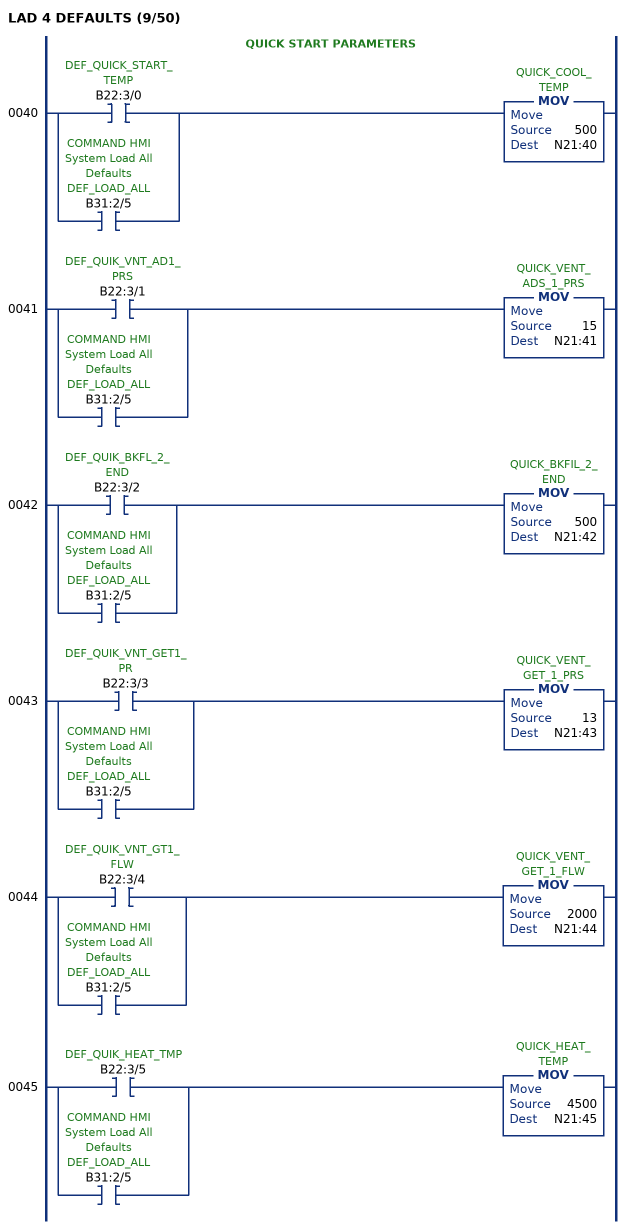
% Rung: 40 %
% TITLE: QUICK START PARAMETERS %
SOR BST XIC B22:3/0 NXB XIC B31:2/5 BND MOV 500 N21:40 EOR
%   B22:3/0  DEF_QUICK_START_TEMP %
%   B31:2/5  DEF_LOAD_ALL  "COMMAND HMI System Load All Defaults" %
%   N21:40  QUICK_COOL_TEMP %
% Rung: 41 %
SOR BST XIC B22:3/1 NXB XIC B31:2/5 BND MOV 15 N21:41 EOR
%   B22:3/1  DEF_QUIK_VNT_AD1_PRS %
%   B31:2/5  DEF_LOAD_ALL  "COMMAND HMI System Load All Defaults" %
%   N21:41  QUICK_VENT_ADS_1_PRS %
% Rung: 42 %
SOR BST XIC B22:3/2 NXB XIC B31:2/5 BND MOV 500 N21:42 EOR
%   B22:3/2  DEF_QUIK_BKFL_2_END %
%   B31:2/5  DEF_LOAD_ALL  "COMMAND HMI System Load All Defaults" %
%   N21:42  QUICK_BKFIL_2_END %
% Rung: 43 %
SOR BST XIC B22:3/3 NXB XIC B31:2/5 BND MOV 13 N21:43 EOR
%   B22:3/3  DEF_QUIK_VNT_GET1_PR %
%   B31:2/5  DEF_LOAD_ALL  "COMMAND HMI System Load All Defaults" %
%   N21:43  QUICK_VENT_GET_1_PRS %
% Rung: 44 %
SOR BST XIC B22:3/4 NXB XIC B31:2/5 BND MOV 2000 N21:44 EOR
%   B22:3/4  DEF_QUIK_VNT_GT1_FLW %
%   B31:2/5  DEF_LOAD_ALL  "COMMAND HMI System Load All Defaults" %
%   N21:44  QUICK_VENT_GET_1_FLW %
% Rung: 45 %
SOR BST XIC B22:3/5 NXB XIC B31:2/5 BND MOV 4500 N21:45 EOR
%   B22:3/5  DEF_QUIK_HEAT_TMP %
%   B31:2/5  DEF_LOAD_ALL  "COMMAND HMI System Load All Defaults" %
%   N21:45  QUICK_HEAT_TEMP %

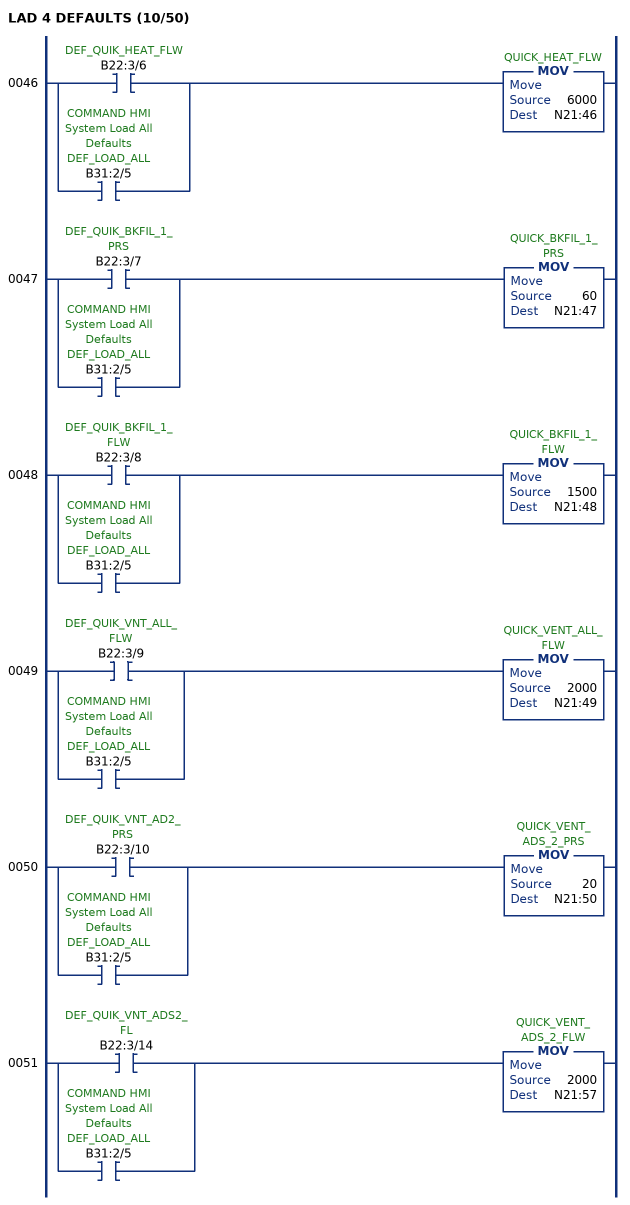
% Rung: 46 %
SOR BST XIC B22:3/6 NXB XIC B31:2/5 BND MOV 6000 N21:46 EOR
%   B22:3/6  DEF_QUIK_HEAT_FLW %
%   B31:2/5  DEF_LOAD_ALL  "COMMAND HMI System Load All Defaults" %
%   N21:46  QUICK_HEAT_FLW %
% Rung: 47 %
SOR BST XIC B22:3/7 NXB XIC B31:2/5 BND MOV 60 N21:47 EOR
%   B22:3/7  DEF_QUIK_BKFIL_1_PRS %
%   B31:2/5  DEF_LOAD_ALL  "COMMAND HMI System Load All Defaults" %
%   N21:47  QUICK_BKFIL_1_PRS %
% Rung: 48 %
SOR BST XIC B22:3/8 NXB XIC B31:2/5 BND MOV 1500 N21:48 EOR
%   B22:3/8  DEF_QUIK_BKFIL_1_FLW %
%   B31:2/5  DEF_LOAD_ALL  "COMMAND HMI System Load All Defaults" %
%   N21:48  QUICK_BKFIL_1_FLW %
% Rung: 49 %
SOR BST XIC B22:3/9 NXB XIC B31:2/5 BND MOV 2000 N21:49 EOR
%   B22:3/9  DEF_QUIK_VNT_ALL_FLW %
%   B31:2/5  DEF_LOAD_ALL  "COMMAND HMI System Load All Defaults" %
%   N21:49  QUICK_VENT_ALL_FLW %
% Rung: 50 %
SOR BST XIC B22:3/10 NXB XIC B31:2/5 BND MOV 20 N21:50 EOR
%   B22:3/10  DEF_QUIK_VNT_AD2_PRS %
%   B31:2/5  DEF_LOAD_ALL  "COMMAND HMI System Load All Defaults" %
%   N21:50  QUICK_VENT_ADS_2_PRS %
% Rung: 51 %
SOR BST XIC B22:3/14 NXB XIC B31:2/5 BND MOV 2000 N21:57 EOR
%   B22:3/14  DEF_QUIK_VNT_ADS2_FL %
%   B31:2/5  DEF_LOAD_ALL  "COMMAND HMI System Load All Defaults" %
%   N21:57  QUICK_VENT_ADS_2_FLW %

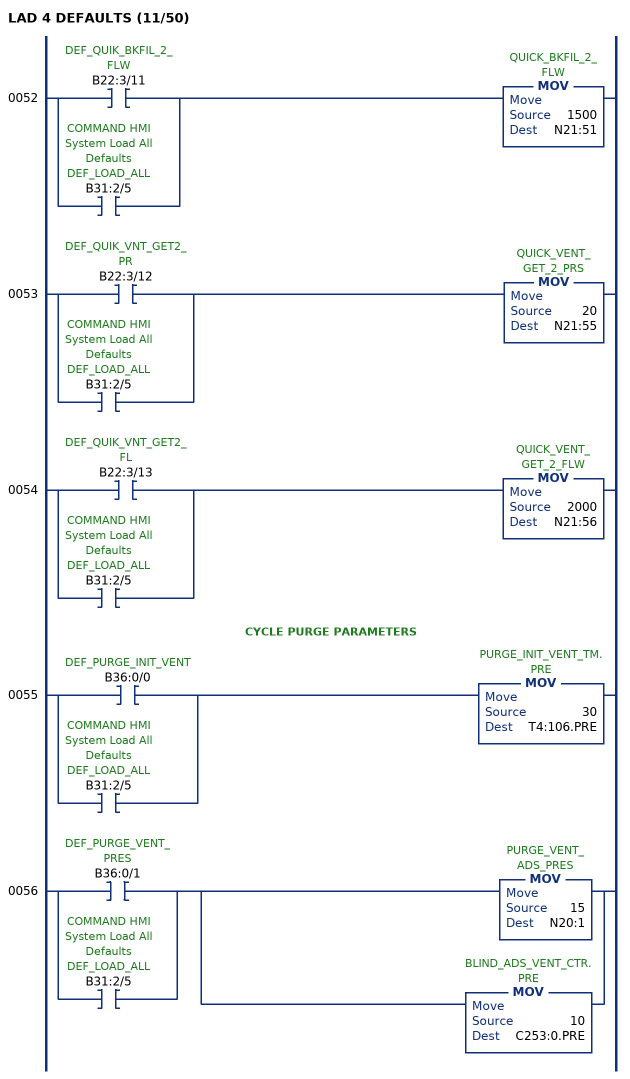
% Rung: 52 %
SOR BST XIC B22:3/11 NXB XIC B31:2/5 BND MOV 1500 N21:51 EOR
%   B22:3/11  DEF_QUIK_BKFIL_2_FLW %
%   B31:2/5  DEF_LOAD_ALL  "COMMAND HMI System Load All Defaults" %
%   N21:51  QUICK_BKFIL_2_FLW %
% Rung: 53 %
SOR BST XIC B22:3/12 NXB XIC B31:2/5 BND MOV 20 N21:55 EOR
%   B22:3/12  DEF_QUIK_VNT_GET2_PR %
%   B31:2/5  DEF_LOAD_ALL  "COMMAND HMI System Load All Defaults" %
%   N21:55  QUICK_VENT_GET_2_PRS %
% Rung: 54 %
SOR BST XIC B22:3/13 NXB XIC B31:2/5 BND MOV 2000 N21:56 EOR
%   B22:3/13  DEF_QUIK_VNT_GET2_FL %
%   B31:2/5  DEF_LOAD_ALL  "COMMAND HMI System Load All Defaults" %
%   N21:56  QUICK_VENT_GET_2_FLW %
% Rung: 55 %
% TITLE: CYCLE PURGE PARAMETERS %
SOR BST XIC B36:0/0 NXB XIC B31:2/5 BND MOV 30 T4:106.PRE EOR
%   B36:0/0  DEF_PURGE_INIT_VENT %
%   B31:2/5  DEF_LOAD_ALL  "COMMAND HMI System Load All Defaults" %
%   T4:106  PURGE_INIT_VENT_TM %
% Rung: 56 %
SOR BST XIC B36:0/1 NXB XIC B31:2/5 BND BST MOV 15 N20:1 NXB MOV 10 C253:0.PRE BND EOR
%   B36:0/1  DEF_PURGE_VENT_PRES %
%   B31:2/5  DEF_LOAD_ALL  "COMMAND HMI System Load All Defaults" %
%   N20:1  PURGE_VENT_ADS_PRES %
%   C253:0  BLIND_ADS_VENT_CTR %

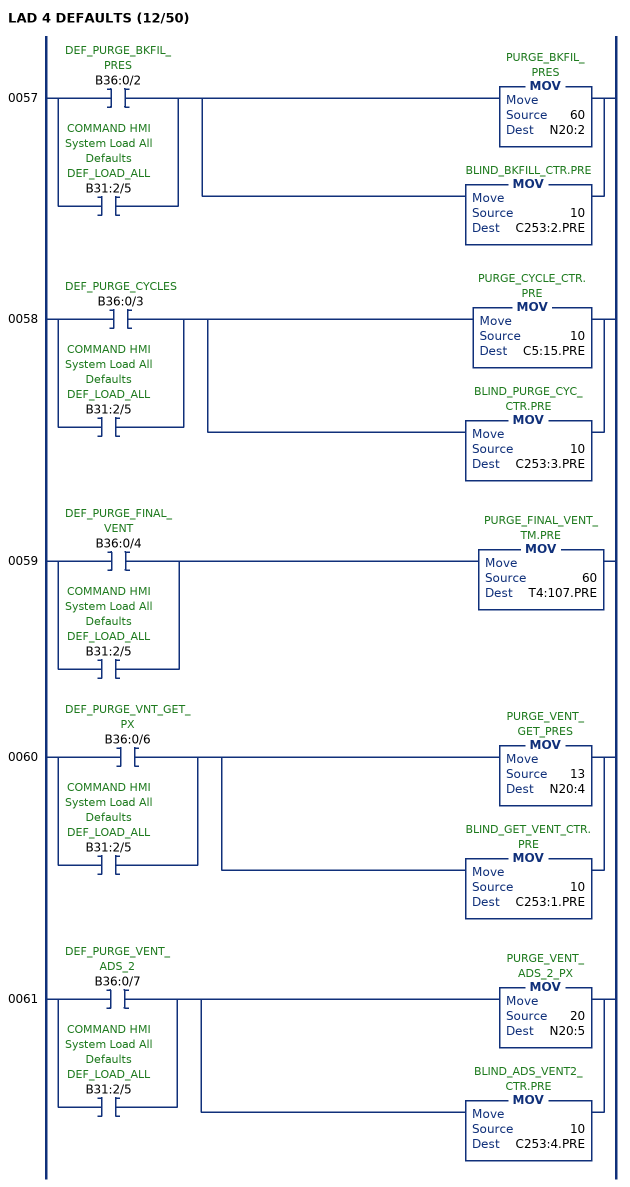
% Rung: 57 %
SOR BST XIC B36:0/2 NXB XIC B31:2/5 BND BST MOV 60 N20:2 NXB MOV 10 C253:2.PRE BND EOR
%   B36:0/2  DEF_PURGE_BKFIL_PRES %
%   B31:2/5  DEF_LOAD_ALL  "COMMAND HMI System Load All Defaults" %
%   N20:2  PURGE_BKFIL_PRES %
%   C253:2  BLIND_BKFILL_CTR %
% Rung: 58 %
SOR BST XIC B36:0/3 NXB XIC B31:2/5 BND BST MOV 10 C5:15.PRE NXB MOV 10 C253:3.PRE BND EOR
%   B36:0/3  DEF_PURGE_CYCLES %
%   B31:2/5  DEF_LOAD_ALL  "COMMAND HMI System Load All Defaults" %
%   C5:15  PURGE_CYCLE_CTR %
%   C253:3  BLIND_PURGE_CYC_CTR %
% Rung: 59 %
SOR BST XIC B36:0/4 NXB XIC B31:2/5 BND MOV 60 T4:107.PRE EOR
%   B36:0/4  DEF_PURGE_FINAL_VENT %
%   B31:2/5  DEF_LOAD_ALL  "COMMAND HMI System Load All Defaults" %
%   T4:107  PURGE_FINAL_VENT_TM %
% Rung: 60 %
SOR BST XIC B36:0/6 NXB XIC B31:2/5 BND BST MOV 13 N20:4 NXB MOV 10 C253:1.PRE BND EOR
%   B36:0/6  DEF_PURGE_VNT_GET_PX %
%   B31:2/5  DEF_LOAD_ALL  "COMMAND HMI System Load All Defaults" %
%   N20:4  PURGE_VENT_GET_PRES %
%   C253:1  BLIND_GET_VENT_CTR %
% Rung: 61 %
SOR BST XIC B36:0/7 NXB XIC B31:2/5 BND BST MOV 20 N20:5 NXB MOV 10 C253:4.PRE BND EOR
%   B36:0/7  DEF_PURGE_VENT_ADS_2 %
%   B31:2/5  DEF_LOAD_ALL  "COMMAND HMI System Load All Defaults" %
%   N20:5  PURGE_VENT_ADS_2_PX %
%   C253:4  BLIND_ADS_VENT2_CTR %

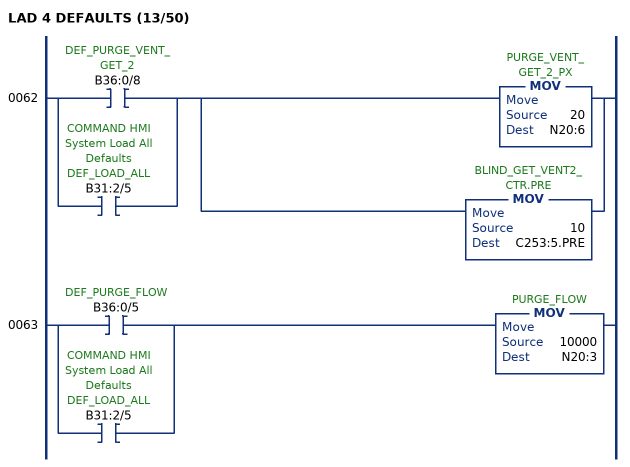
% Rung: 62 %
SOR BST XIC B36:0/8 NXB XIC B31:2/5 BND BST MOV 20 N20:6 NXB MOV 10 C253:5.PRE BND EOR
%   B36:0/8  DEF_PURGE_VENT_GET_2 %
%   B31:2/5  DEF_LOAD_ALL  "COMMAND HMI System Load All Defaults" %
%   N20:6  PURGE_VENT_GET_2_PX %
%   C253:5  BLIND_GET_VENT2_CTR %
% Rung: 63 %
SOR BST XIC B36:0/5 NXB XIC B31:2/5 BND MOV 10000 N20:3 EOR
%   B36:0/5  DEF_PURGE_FLOW %
%   B31:2/5  DEF_LOAD_ALL  "COMMAND HMI System Load All Defaults" %
%   N20:3  PURGE_FLOW %

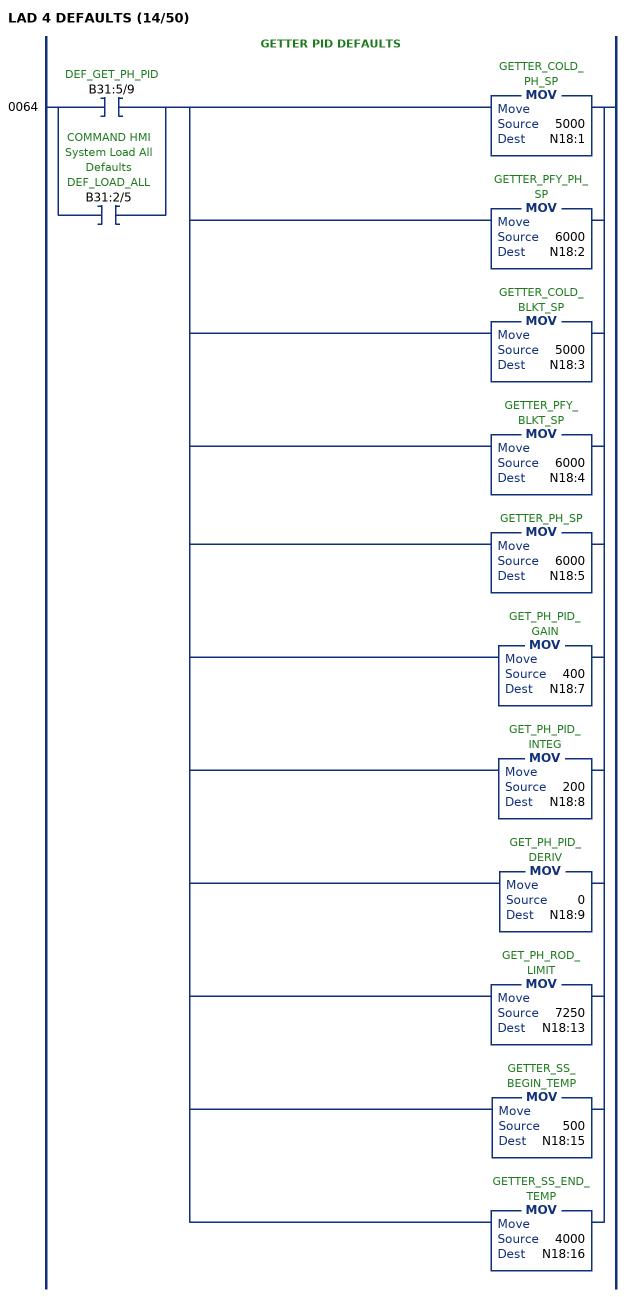
% Rung: 64 %
% TITLE: GETTER PID DEFAULTS %
SOR BST XIC B31:5/9 NXB XIC B31:2/5 BND BST MOV 5000 N18:1 NXB MOV 6000 N18:2 NXB MOV 5000 N18:3 NXB MOV 6000 N18:4 NXB MOV 6000 N18:5 NXB MOV 400 N18:7 NXB MOV 200 N18:8 NXB MOV 0 N18:9 NXB MOV 7250 N18:13 NXB MOV 500 N18:15 NXB MOV 4000 N18:16 BND EOR
%   B31:5/9  DEF_GET_PH_PID %
%   B31:2/5  DEF_LOAD_ALL  "COMMAND HMI System Load All Defaults" %
%   N18:1  GETTER_COLD_PH_SP %
%   N18:2  GETTER_PFY_PH_SP %
%   N18:3  GETTER_COLD_BLKT_SP %
%   N18:4  GETTER_PFY_BLKT_SP %
%   N18:5  GETTER_PH_SP %
%   N18:7  GET_PH_PID_GAIN %
%   N18:8  GET_PH_PID_INTEG %
%   N18:9  GET_PH_PID_DERIV %
%   N18:13  GET_PH_ROD_LIMIT %
%   N18:15  GETTER_SS_BEGIN_TEMP %
%   N18:16  GETTER_SS_END_TEMP %

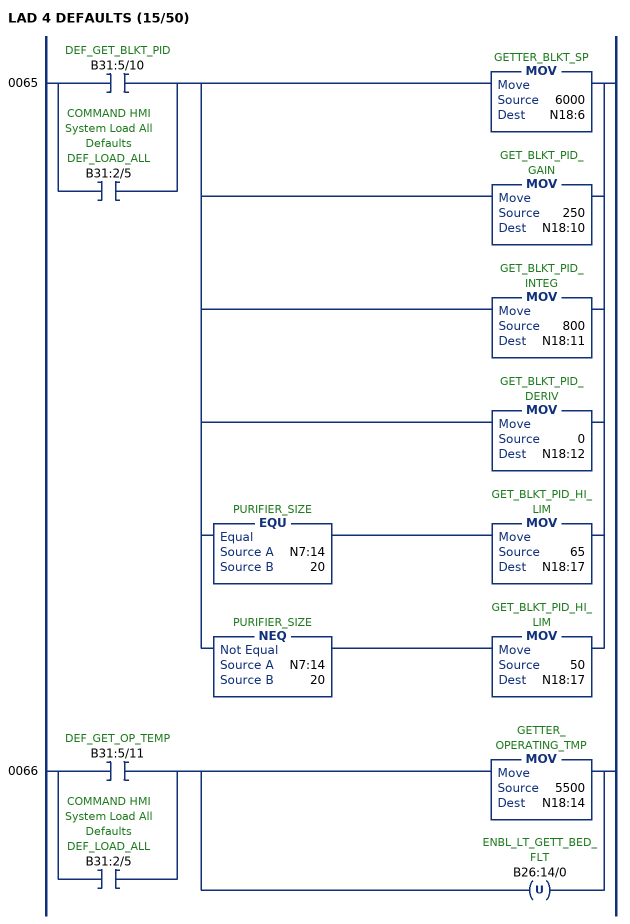
% Rung: 65 %
SOR BST XIC B31:5/10 NXB XIC B31:2/5 BND BST MOV 6000 N18:6 NXB MOV 250 N18:10 NXB MOV 800 N18:11 NXB MOV 0 N18:12 NXB EQU N7:14 20 MOV 65 N18:17 NXB NEQ N7:14 20 MOV 50 N18:17 BND EOR
%   B31:5/10  DEF_GET_BLKT_PID %
%   B31:2/5  DEF_LOAD_ALL  "COMMAND HMI System Load All Defaults" %
%   N18:6  GETTER_BLKT_SP %
%   N18:10  GET_BLKT_PID_GAIN %
%   N18:11  GET_BLKT_PID_INTEG %
%   N18:12  GET_BLKT_PID_DERIV %
%   N7:14  PURIFIER_SIZE %
%   N18:17  GET_BLKT_PID_HI_LIM %
% Rung: 66 %
SOR BST XIC B31:5/11 NXB XIC B31:2/5 BND BST MOV 5500 N18:14 NXB OTU B26:14/0 BND EOR
%   B31:5/11  DEF_GET_OP_TEMP %
%   B31:2/5  DEF_LOAD_ALL  "COMMAND HMI System Load All Defaults" %
%   N18:14  GETTER_OPERATING_TMP %
%   B26:14/0  ENBL_LT_GETT_BED_FLT %

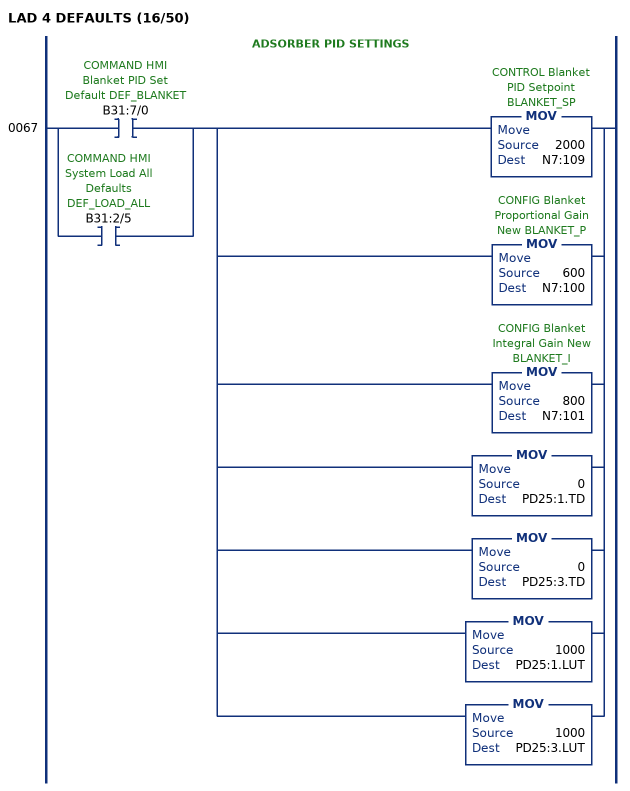
% Rung: 67 %
% TITLE: ADSORBER PID SETTINGS %
SOR BST XIC B31:7/0 NXB XIC B31:2/5 BND BST MOV 2000 N7:109 NXB MOV 600 N7:100 NXB MOV 800 N7:101 NXB MOV 0 PD25:1.TD NXB MOV 0 PD25:3.TD NXB MOV 1000 PD25:1.LUT NXB MOV 1000 PD25:3.LUT BND EOR
%   B31:7/0  DEF_BLANKET  "COMMAND HMI Blanket PID Set Default" %
%   B31:2/5  DEF_LOAD_ALL  "COMMAND HMI System Load All Defaults" %
%   N7:109  BLANKET_SP  "CONTROL Blanket PID Setpoint" %
%   N7:100  BLANKET_P  "CONFIG Blanket Proportional Gain New" %
%   N7:101  BLANKET_I  "CONFIG Blanket Integral Gain New" %

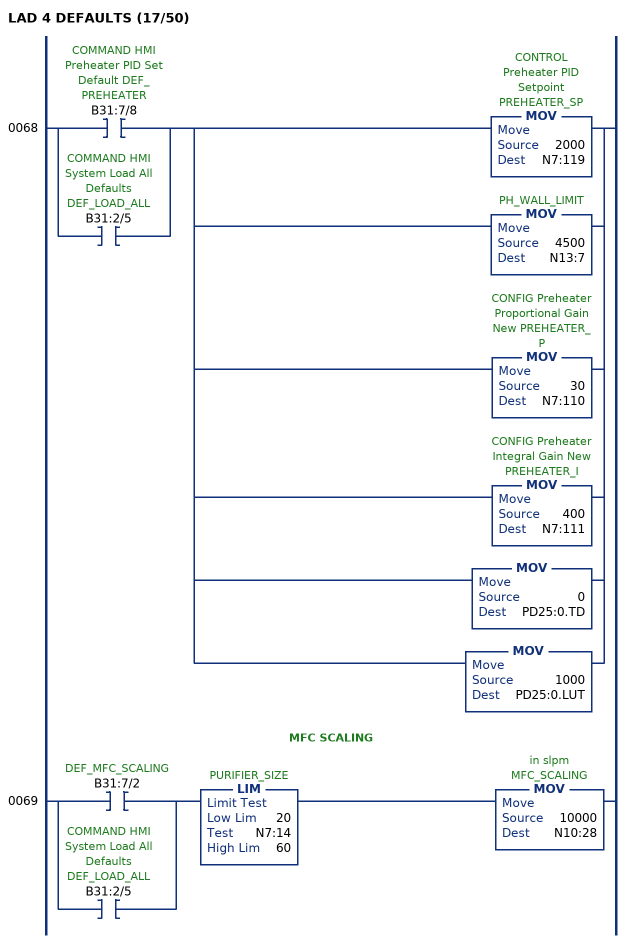
% Rung: 68 %
SOR BST XIC B31:7/8 NXB XIC B31:2/5 BND BST MOV 2000 N7:119 NXB MOV 4500 N13:7 NXB MOV 30 N7:110 NXB MOV 400 N7:111 NXB MOV 0 PD25:0.TD NXB MOV 1000 PD25:0.LUT BND EOR
%   B31:7/8  DEF_PREHEATER  "COMMAND HMI Preheater PID Set Default" %
%   B31:2/5  DEF_LOAD_ALL  "COMMAND HMI System Load All Defaults" %
%   N7:119  PREHEATER_SP  "CONTROL Preheater PID Setpoint" %
%   N13:7  PH_WALL_LIMIT %
%   N7:110  PREHEATER_P  "CONFIG Preheater Proportional Gain New" %
%   N7:111  PREHEATER_I  "CONFIG Preheater Integral Gain New" %
% Rung: 69 %
% TITLE: MFC SCALING %
SOR BST XIC B31:7/2 NXB XIC B31:2/5 BND LIM 20 N7:14 60 MOV 10000 N10:28 EOR
%   B31:7/2  DEF_MFC_SCALING %
%   B31:2/5  DEF_LOAD_ALL  "COMMAND HMI System Load All Defaults" %
%   N7:14  PURIFIER_SIZE %
%   N10:28  MFC_SCALING  "in slpm" %

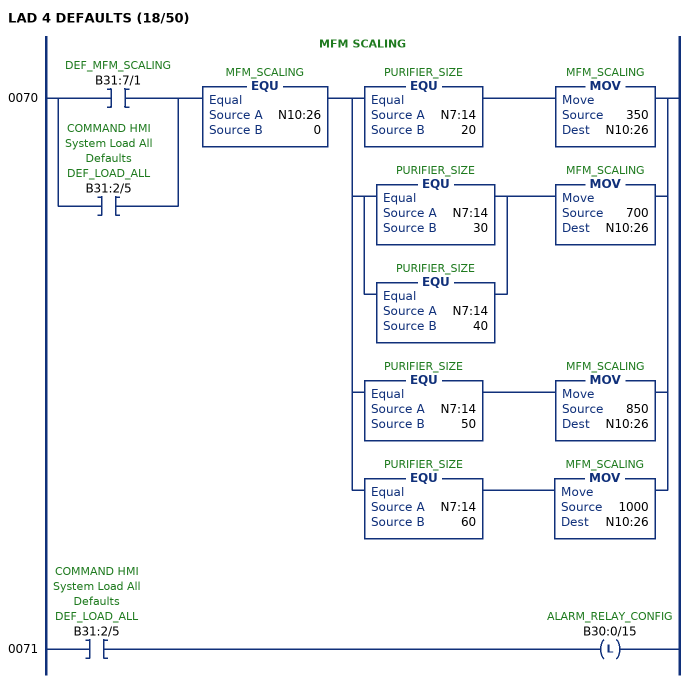
% Rung: 70 %
% TITLE: MFM SCALING %
SOR BST XIC B31:7/1 NXB XIC B31:2/5 BND EQU N10:26 0 BST EQU N7:14 20 MOV 350 N10:26 NXB BST EQU N7:14 30 NXB EQU N7:14 40 BND MOV 700 N10:26 NXB EQU N7:14 50 MOV 850 N10:26 NXB EQU N7:14 60 MOV 1000 N10:26 BND EOR
%   B31:7/1  DEF_MFM_SCALING %
%   B31:2/5  DEF_LOAD_ALL  "COMMAND HMI System Load All Defaults" %
%   N10:26  MFM_SCALING %
%   N7:14  PURIFIER_SIZE %
% Rung: 71 %
SOR XIC B31:2/5 OTL B30:0/15 EOR
%   B31:2/5  DEF_LOAD_ALL  "COMMAND HMI System Load All Defaults" %
%   B30:0/15  ALARM_RELAY_CONFIG %

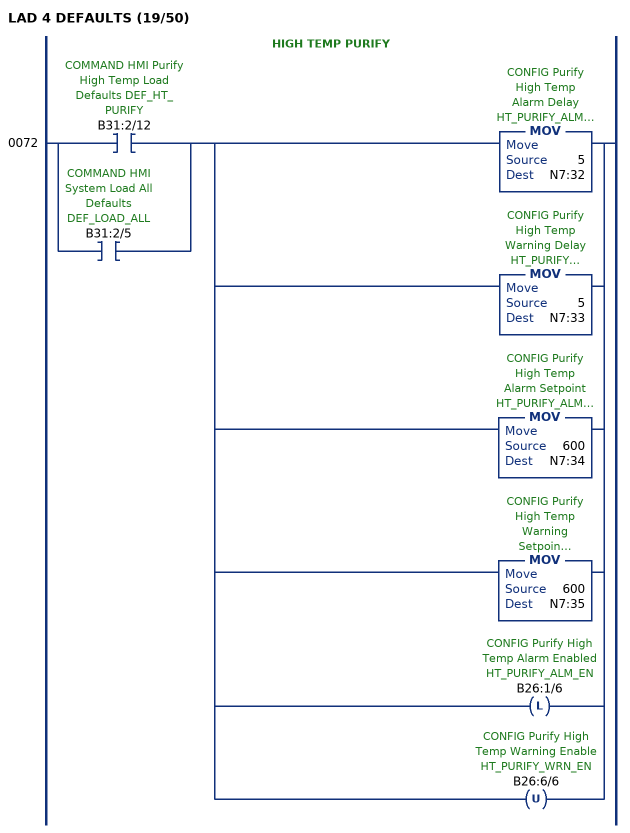
% Rung: 72 %
% TITLE: HIGH TEMP PURIFY %
SOR BST XIC B31:2/12 NXB XIC B31:2/5 BND BST MOV 5 N7:32 NXB MOV 5 N7:33 NXB MOV 600 N7:34 NXB MOV 600 N7:35 NXB OTL B26:1/6 NXB OTU B26:6/6 BND EOR
%   B31:2/12  DEF_HT_PURIFY  "COMMAND HMI Purify High Temp Load Defaults" %
%   B31:2/5  DEF_LOAD_ALL  "COMMAND HMI System Load All Defaults" %
%   N7:32  HT_PURIFY_ALM_DLY  "CONFIG Purify High Temp Alarm Delay" %
%   N7:33  HT_PURIFY_WRN_DLY  "CONFIG Purify High Temp Warning Delay" %
%   N7:34  HT_PURIFY_ALM_SP  "CONFIG Purify High Temp Alarm Setpoint" %
%   N7:35  HT_PURIFY_WRN_SP  "CONFIG Purify High Temp Warning Setpoint" %
%   B26:1/6  HT_PURIFY_ALM_EN  "CONFIG Purify High Temp Alarm Enabled" %
%   B26:6/6  HT_PURIFY_WRN_EN  "CONFIG Purify High Temp Warning Enable" %

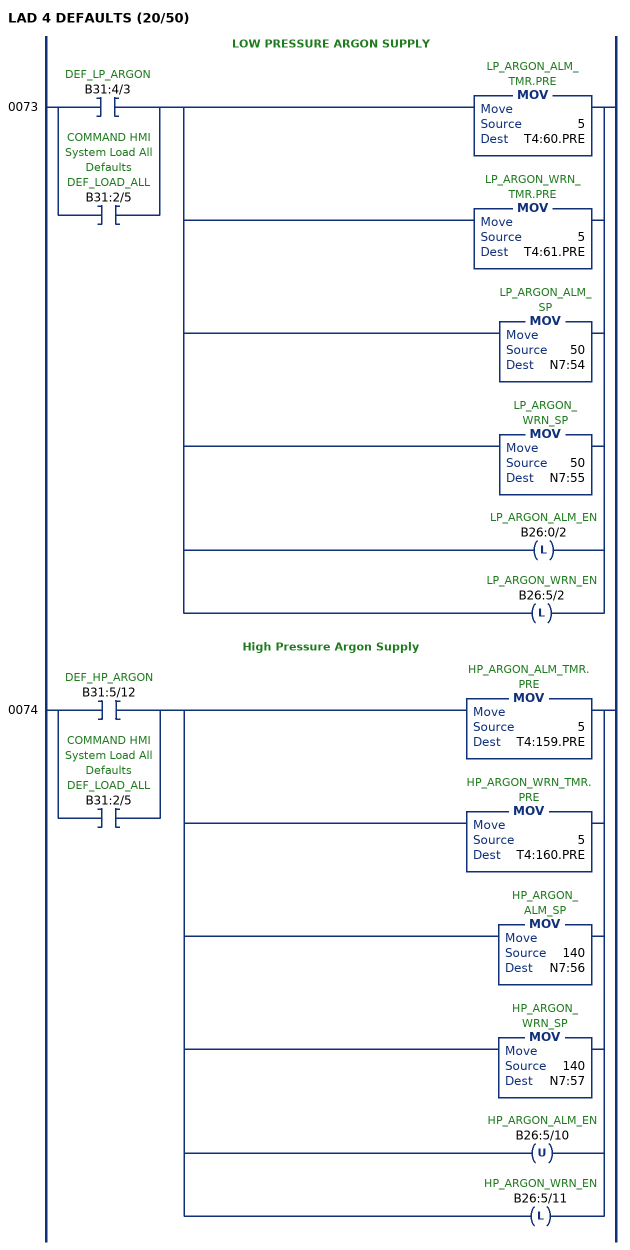
% Rung: 73 %
% TITLE: LOW PRESSURE ARGON SUPPLY %
SOR BST XIC B31:4/3 NXB XIC B31:2/5 BND BST MOV 5 T4:60.PRE NXB MOV 5 T4:61.PRE NXB MOV 50 N7:54 NXB MOV 50 N7:55 NXB OTL B26:0/2 NXB OTL B26:5/2 BND EOR
%   B31:4/3  DEF_LP_ARGON %
%   B31:2/5  DEF_LOAD_ALL  "COMMAND HMI System Load All Defaults" %
%   T4:60  LP_ARGON_ALM_TMR %
%   T4:61  LP_ARGON_WRN_TMR %
%   N7:54  LP_ARGON_ALM_SP %
%   N7:55  LP_ARGON_WRN_SP %
%   B26:0/2  LP_ARGON_ALM_EN %
%   B26:5/2  LP_ARGON_WRN_EN %
% Rung: 74 %
% TITLE: High Pressure Argon Supply %
SOR BST XIC B31:5/12 NXB XIC B31:2/5 BND BST MOV 5 T4:159.PRE NXB MOV 5 T4:160.PRE NXB MOV 140 N7:56 NXB MOV 140 N7:57 NXB OTU B26:5/10 NXB OTL B26:5/11 BND EOR
%   B31:5/12  DEF_HP_ARGON %
%   B31:2/5  DEF_LOAD_ALL  "COMMAND HMI System Load All Defaults" %
%   T4:159  HP_ARGON_ALM_TMR %
%   T4:160  HP_ARGON_WRN_TMR %
%   N7:56  HP_ARGON_ALM_SP %
%   N7:57  HP_ARGON_WRN_SP %
%   B26:5/10  HP_ARGON_ALM_EN %
%   B26:5/11  HP_ARGON_WRN_EN %

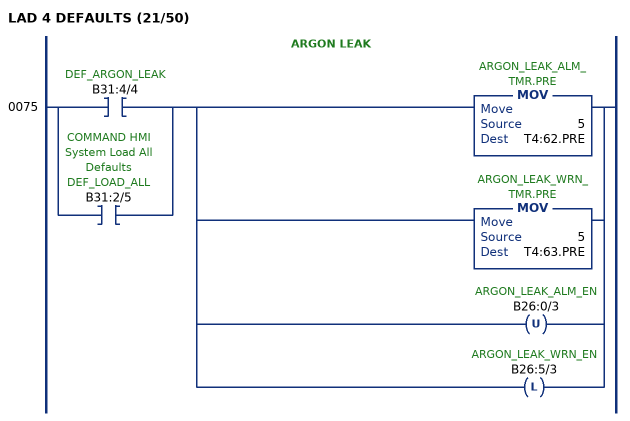
% Rung: 75 %
% TITLE: ARGON LEAK %
SOR BST XIC B31:4/4 NXB XIC B31:2/5 BND BST MOV 5 T4:62.PRE NXB MOV 5 T4:63.PRE NXB OTU B26:0/3 NXB OTL B26:5/3 BND EOR
%   B31:4/4  DEF_ARGON_LEAK %
%   B31:2/5  DEF_LOAD_ALL  "COMMAND HMI System Load All Defaults" %
%   T4:62  ARGON_LEAK_ALM_TMR %
%   T4:63  ARGON_LEAK_WRN_TMR %
%   B26:0/3  ARGON_LEAK_ALM_EN %
%   B26:5/3  ARGON_LEAK_WRN_EN %

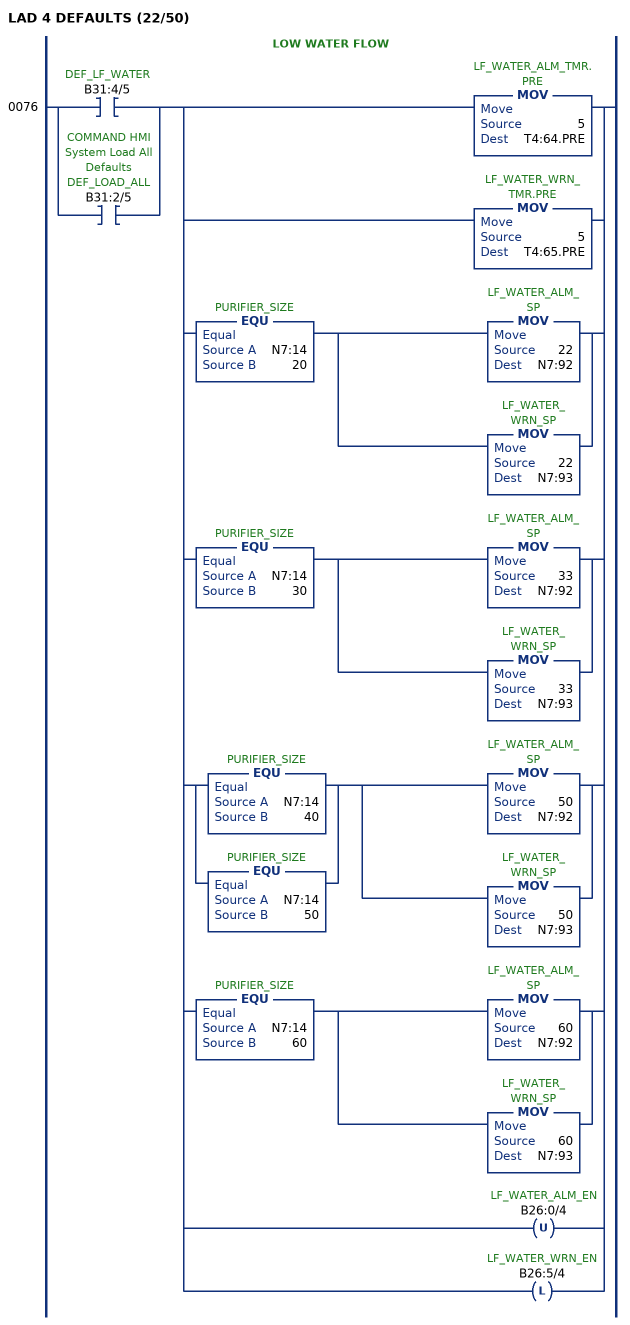
% Rung: 76 %
% TITLE: LOW WATER FLOW %
SOR BST XIC B31:4/5 NXB XIC B31:2/5 BND BST MOV 5 T4:64.PRE NXB MOV 5 T4:65.PRE NXB EQU N7:14 20 BST MOV 22 N7:92 NXB MOV 22 N7:93 BND NXB EQU N7:14 30 BST MOV 33 N7:92 NXB MOV 33 N7:93 BND NXB BST EQU N7:14 40 NXB EQU N7:14 50 BND BST MOV 50 N7:92 NXB MOV 50 N7:93 BND NXB EQU N7:14 60 BST MOV 60 N7:92 NXB MOV 60 N7:93 BND NXB OTU B26:0/4 NXB OTL B26:5/4 BND EOR
%   B31:4/5  DEF_LF_WATER %
%   B31:2/5  DEF_LOAD_ALL  "COMMAND HMI System Load All Defaults" %
%   T4:64  LF_WATER_ALM_TMR %
%   T4:65  LF_WATER_WRN_TMR %
%   N7:14  PURIFIER_SIZE %
%   N7:92  LF_WATER_ALM_SP %
%   N7:93  LF_WATER_WRN_SP %
%   B26:0/4  LF_WATER_ALM_EN %
%   B26:5/4  LF_WATER_WRN_EN %

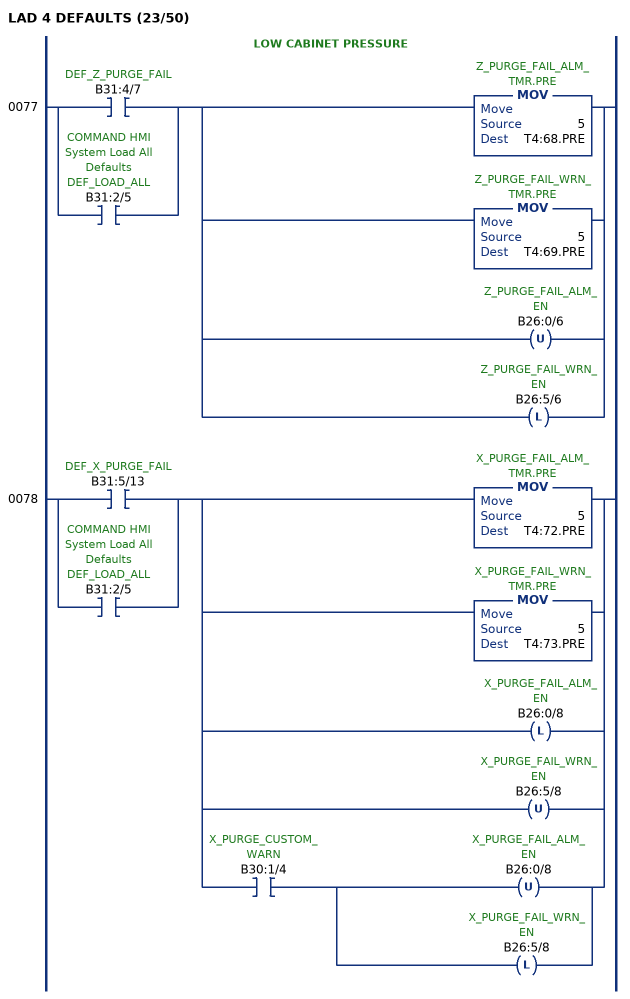
% Rung: 77 %
% TITLE: LOW CABINET PRESSURE %
SOR BST XIC B31:4/7 NXB XIC B31:2/5 BND BST MOV 5 T4:68.PRE NXB MOV 5 T4:69.PRE NXB OTU B26:0/6 NXB OTL B26:5/6 BND EOR
%   B31:4/7  DEF_Z_PURGE_FAIL %
%   B31:2/5  DEF_LOAD_ALL  "COMMAND HMI System Load All Defaults" %
%   T4:68  Z_PURGE_FAIL_ALM_TMR %
%   T4:69  Z_PURGE_FAIL_WRN_TMR %
%   B26:0/6  Z_PURGE_FAIL_ALM_EN %
%   B26:5/6  Z_PURGE_FAIL_WRN_EN %
% Rung: 78 %
SOR BST XIC B31:5/13 NXB XIC B31:2/5 BND BST MOV 5 T4:72.PRE NXB MOV 5 T4:73.PRE NXB BST OTL B26:0/8 NXB OTU B26:5/8 BND NXB XIC B30:1/4 BST OTU B26:0/8 NXB OTL B26:5/8 BND BND EOR
%   B31:5/13  DEF_X_PURGE_FAIL %
%   B31:2/5  DEF_LOAD_ALL  "COMMAND HMI System Load All Defaults" %
%   T4:72  X_PURGE_FAIL_ALM_TMR %
%   T4:73  X_PURGE_FAIL_WRN_TMR %
%   B26:0/8  X_PURGE_FAIL_ALM_EN %
%   B26:5/8  X_PURGE_FAIL_WRN_EN %
%   B30:1/4  X_PURGE_CUSTOM_WARN %

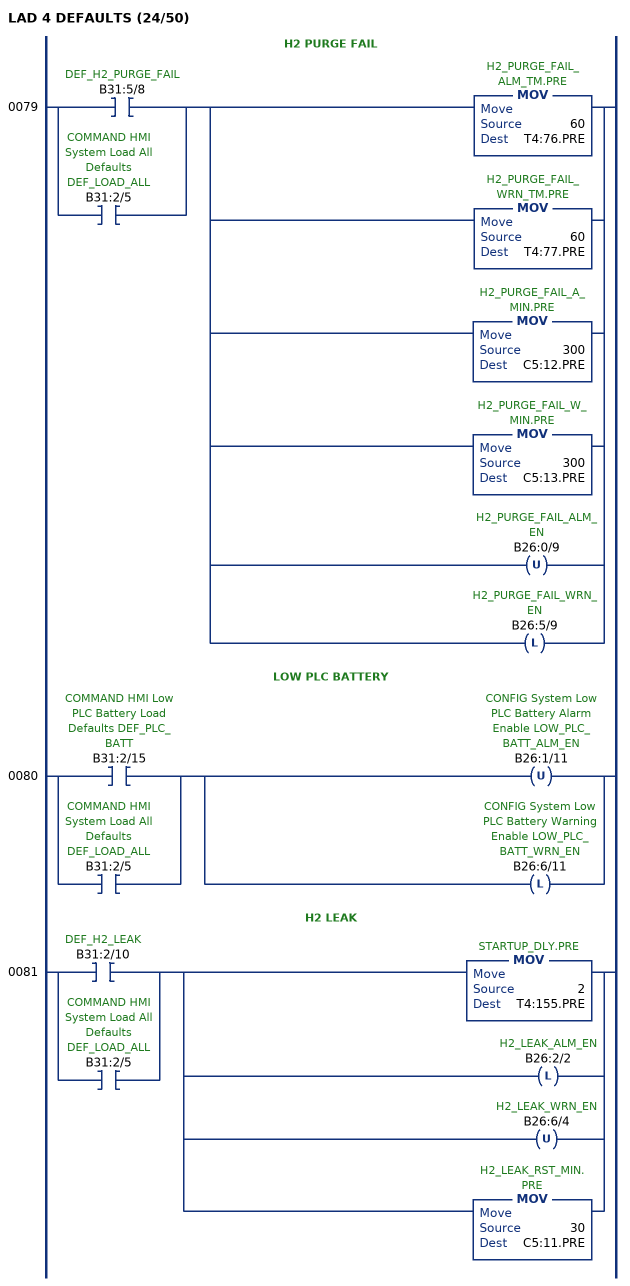
% Rung: 79 %
% TITLE: H2 PURGE FAIL %
SOR BST XIC B31:5/8 NXB XIC B31:2/5 BND BST MOV 60 T4:76.PRE NXB MOV 60 T4:77.PRE NXB MOV 300 C5:12.PRE NXB MOV 300 C5:13.PRE NXB OTU B26:0/9 NXB OTL B26:5/9 BND EOR
%   B31:5/8  DEF_H2_PURGE_FAIL %
%   B31:2/5  DEF_LOAD_ALL  "COMMAND HMI System Load All Defaults" %
%   T4:76  H2_PURGE_FAIL_ALM_TM %
%   T4:77  H2_PURGE_FAIL_WRN_TM %
%   C5:12  H2_PURGE_FAIL_A_MIN %
%   C5:13  H2_PURGE_FAIL_W_MIN %
%   B26:0/9  H2_PURGE_FAIL_ALM_EN %
%   B26:5/9  H2_PURGE_FAIL_WRN_EN %
% Rung: 80 %
% TITLE: LOW PLC BATTERY %
SOR BST XIC B31:2/15 NXB XIC B31:2/5 BND BST OTU B26:1/11 NXB OTL B26:6/11 BND EOR
%   B31:2/15  DEF_PLC_BATT  "COMMAND HMI Low PLC Battery Load Defaults" %
%   B31:2/5  DEF_LOAD_ALL  "COMMAND HMI System Load All Defaults" %
%   B26:1/11  LOW_PLC_BATT_ALM_EN  "CONFIG System Low PLC Battery Alarm Enable" %
%   B26:6/11  LOW_PLC_BATT_WRN_EN  "CONFIG System Low PLC Battery Warning Enable" %
% Rung: 81 %
% TITLE: H2 LEAK %
SOR BST XIC B31:2/10 NXB XIC B31:2/5 BND BST MOV 2 T4:155.PRE NXB OTL B26:2/2 NXB OTU B26:6/4 NXB MOV 30 C5:11.PRE BND EOR
%   B31:2/10  DEF_H2_LEAK %
%   B31:2/5  DEF_LOAD_ALL  "COMMAND HMI System Load All Defaults" %
%   T4:155  STARTUP_DLY %
%   B26:2/2  H2_LEAK_ALM_EN %
%   B26:6/4  H2_LEAK_WRN_EN %
%   C5:11  H2_LEAK_RST_MIN %

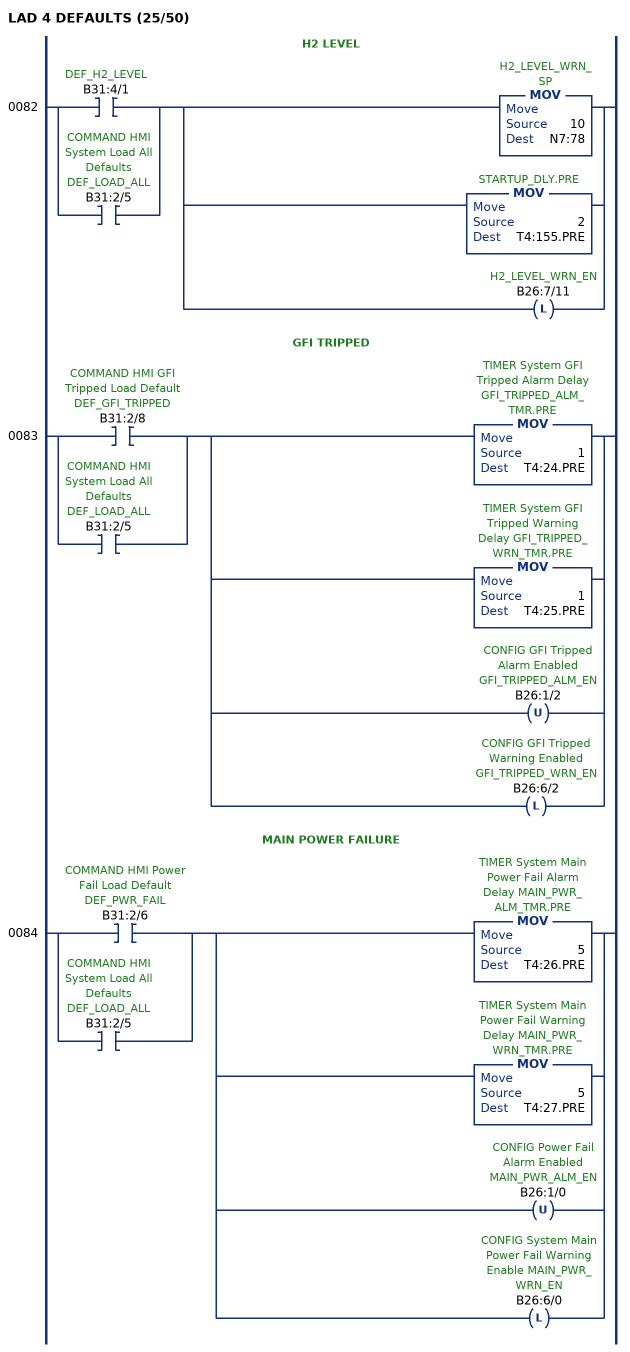
% Rung: 82 %
% TITLE: H2 LEVEL %
SOR BST XIC B31:4/1 NXB XIC B31:2/5 BND BST MOV 10 N7:78 NXB MOV 2 T4:155.PRE NXB OTL B26:7/11 BND EOR
%   B31:4/1  DEF_H2_LEVEL %
%   B31:2/5  DEF_LOAD_ALL  "COMMAND HMI System Load All Defaults" %
%   N7:78  H2_LEVEL_WRN_SP %
%   T4:155  STARTUP_DLY %
%   B26:7/11  H2_LEVEL_WRN_EN %
% Rung: 83 %
% TITLE: GFI TRIPPED %
SOR BST XIC B31:2/8 NXB XIC B31:2/5 BND BST MOV 1 T4:24.PRE NXB MOV 1 T4:25.PRE NXB OTU B26:1/2 NXB OTL B26:6/2 BND EOR
%   B31:2/8  DEF_GFI_TRIPPED  "COMMAND HMI GFI Tripped Load Default" %
%   B31:2/5  DEF_LOAD_ALL  "COMMAND HMI System Load All Defaults" %
%   T4:24  GFI_TRIPPED_ALM_TMR  "TIMER System GFI Tripped Alarm Delay" %
%   T4:25  GFI_TRIPPED_WRN_TMR  "TIMER System GFI Tripped Warning Delay" %
%   B26:1/2  GFI_TRIPPED_ALM_EN  "CONFIG GFI Tripped Alarm Enabled" %
%   B26:6/2  GFI_TRIPPED_WRN_EN  "CONFIG GFI Tripped Warning Enabled" %
% Rung: 84 %
% TITLE: MAIN POWER FAILURE %
SOR BST XIC B31:2/6 NXB XIC B31:2/5 BND BST MOV 5 T4:26.PRE NXB MOV 5 T4:27.PRE NXB OTU B26:1/0 NXB OTL B26:6/0 BND EOR
%   B31:2/6  DEF_PWR_FAIL  "COMMAND HMI Power Fail Load Default" %
%   B31:2/5  DEF_LOAD_ALL  "COMMAND HMI System Load All Defaults" %
%   T4:26  MAIN_PWR_ALM_TMR  "TIMER System Main Power Fail Alarm Delay" %
%   T4:27  MAIN_PWR_WRN_TMR  "TIMER System Main Power Fail Warning Delay" %
%   B26:1/0  MAIN_PWR_ALM_EN  "CONFIG Power Fail Alarm Enabled" %
%   B26:6/0  MAIN_PWR_WRN_EN  "CONFIG System Main Power Fail Warning Enable" %

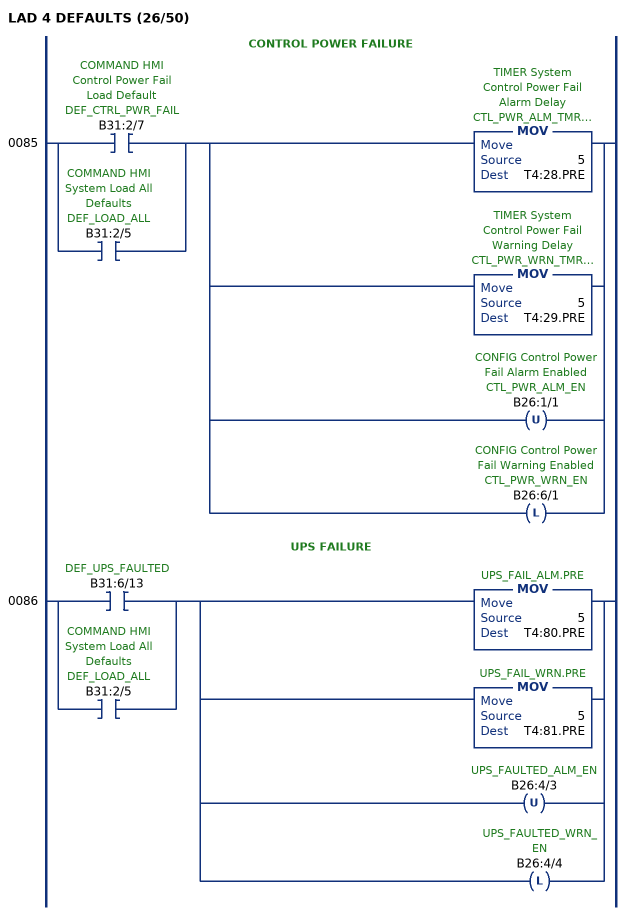
% Rung: 85 %
% TITLE: CONTROL POWER FAILURE %
SOR BST XIC B31:2/7 NXB XIC B31:2/5 BND BST MOV 5 T4:28.PRE NXB MOV 5 T4:29.PRE NXB OTU B26:1/1 NXB OTL B26:6/1 BND EOR
%   B31:2/7  DEF_CTRL_PWR_FAIL  "COMMAND HMI Control Power Fail Load Default" %
%   B31:2/5  DEF_LOAD_ALL  "COMMAND HMI System Load All Defaults" %
%   T4:28  CTL_PWR_ALM_TMR  "TIMER System Control Power Fail Alarm Delay" %
%   T4:29  CTL_PWR_WRN_TMR  "TIMER System Control Power Fail Warning Delay" %
%   B26:1/1  CTL_PWR_ALM_EN  "CONFIG Control Power Fail Alarm Enabled" %
%   B26:6/1  CTL_PWR_WRN_EN  "CONFIG Control Power Fail Warning Enabled" %
% Rung: 86 %
% TITLE: UPS FAILURE %
SOR BST XIC B31:6/13 NXB XIC B31:2/5 BND BST MOV 5 T4:80.PRE NXB MOV 5 T4:81.PRE NXB OTU B26:4/3 NXB OTL B26:4/4 BND EOR
%   B31:6/13  DEF_UPS_FAULTED %
%   B31:2/5  DEF_LOAD_ALL  "COMMAND HMI System Load All Defaults" %
%   T4:80  UPS_FAIL_ALM %
%   T4:81  UPS_FAIL_WRN %
%   B26:4/3  UPS_FAULTED_ALM_EN %
%   B26:4/4  UPS_FAULTED_WRN_EN %

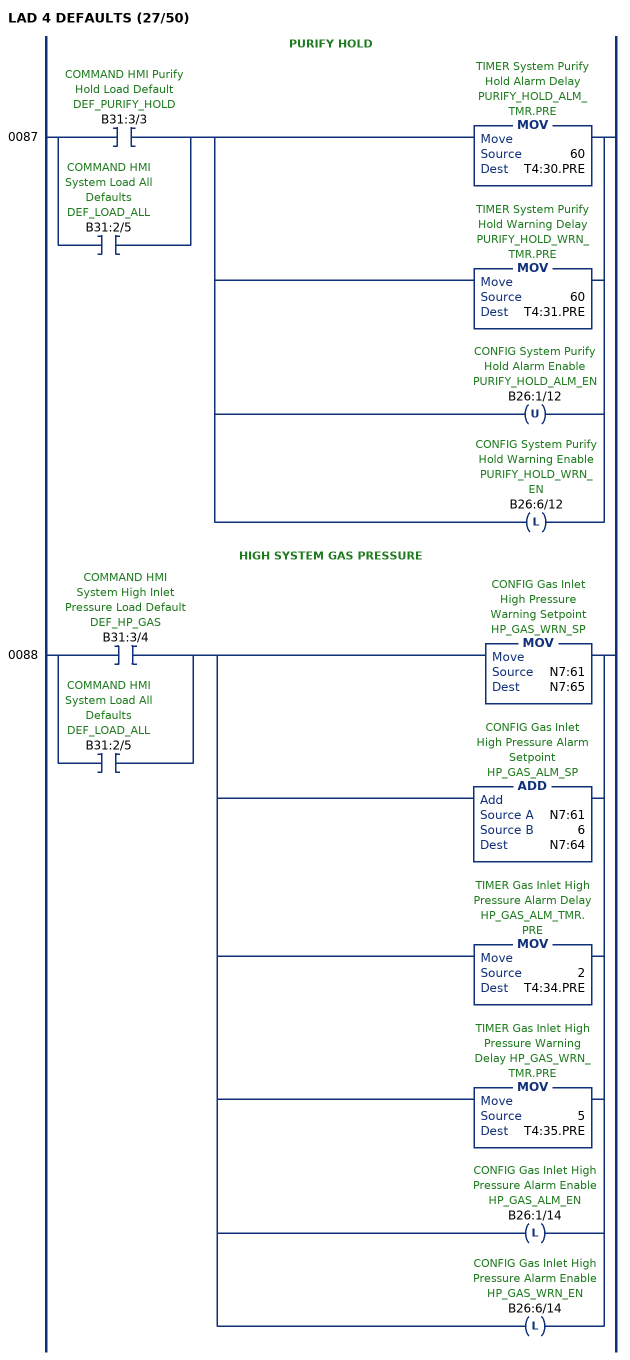
% Rung: 87 %
% TITLE: PURIFY HOLD %
SOR BST XIC B31:3/3 NXB XIC B31:2/5 BND BST MOV 60 T4:30.PRE NXB MOV 60 T4:31.PRE NXB OTU B26:1/12 NXB OTL B26:6/12 BND EOR
%   B31:3/3  DEF_PURIFY_HOLD  "COMMAND HMI Purify Hold Load Default" %
%   B31:2/5  DEF_LOAD_ALL  "COMMAND HMI System Load All Defaults" %
%   T4:30  PURIFY_HOLD_ALM_TMR  "TIMER System Purify Hold Alarm Delay" %
%   T4:31  PURIFY_HOLD_WRN_TMR  "TIMER System Purify Hold Warning Delay" %
%   B26:1/12  PURIFY_HOLD_ALM_EN  "CONFIG System Purify Hold Alarm Enable" %
%   B26:6/12  PURIFY_HOLD_WRN_EN  "CONFIG System Purify Hold Warning Enable" %
% Rung: 88 %
% TITLE: HIGH SYSTEM GAS PRESSURE %
SOR BST XIC B31:3/4 NXB XIC B31:2/5 BND BST MOV N7:61 N7:65 NXB ADD N7:61 6 N7:64 NXB MOV 2 T4:34.PRE NXB MOV 5 T4:35.PRE NXB OTL B26:1/14 NXB OTL B26:6/14 BND EOR
%   B31:3/4  DEF_HP_GAS  "COMMAND HMI System High Inlet Pressure Load Default" %
%   B31:2/5  DEF_LOAD_ALL  "COMMAND HMI System Load All Defaults" %
%   N7:61  HP_GAS_WRN_HMI_SP %
%   N7:65  HP_GAS_WRN_SP  "CONFIG Gas Inlet High Pressure Warning Setpoint" %
%   N7:64  HP_GAS_ALM_SP  "CONFIG Gas Inlet High Pressure Alarm Setpoint" %
%   T4:34  HP_GAS_ALM_TMR  "TIMER Gas Inlet High Pressure Alarm Delay" %
%   T4:35  HP_GAS_WRN_TMR  "TIMER Gas Inlet High Pressure Warning Delay" %
%   B26:1/14  HP_GAS_ALM_EN  "CONFIG Gas Inlet High Pressure Alarm Enable" %
%   B26:6/14  HP_GAS_WRN_EN  "CONFIG Gas Inlet High Pressure Alarm Enable" %

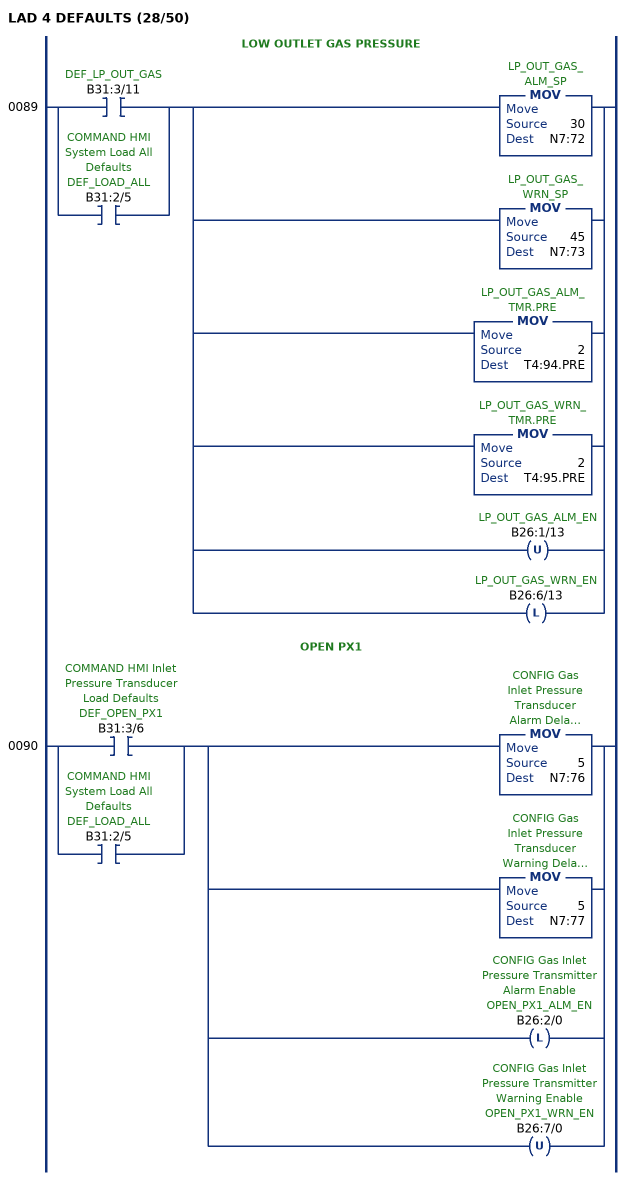
% Rung: 89 %
% TITLE: LOW OUTLET GAS PRESSURE %
SOR BST XIC B31:3/11 NXB XIC B31:2/5 BND BST MOV 30 N7:72 NXB MOV 45 N7:73 NXB MOV 2 T4:94.PRE NXB MOV 2 T4:95.PRE NXB OTU B26:1/13 NXB OTL B26:6/13 BND EOR
%   B31:3/11  DEF_LP_OUT_GAS %
%   B31:2/5  DEF_LOAD_ALL  "COMMAND HMI System Load All Defaults" %
%   N7:72  LP_OUT_GAS_ALM_SP %
%   N7:73  LP_OUT_GAS_WRN_SP %
%   T4:94  LP_OUT_GAS_ALM_TMR %
%   T4:95  LP_OUT_GAS_WRN_TMR %
%   B26:1/13  LP_OUT_GAS_ALM_EN %
%   B26:6/13  LP_OUT_GAS_WRN_EN %
% Rung: 90 %
% TITLE: OPEN PX1 %
SOR BST XIC B31:3/6 NXB XIC B31:2/5 BND BST MOV 5 N7:76 NXB MOV 5 N7:77 NXB OTL B26:2/0 NXB OTU B26:7/0 BND EOR
%   B31:3/6  DEF_OPEN_PX1  "COMMAND HMI Inlet Pressure Transducer Load Defaults" %
%   B31:2/5  DEF_LOAD_ALL  "COMMAND HMI System Load All Defaults" %
%   N7:76  OPEN_PX1_ALM_DLY  "CONFIG Gas Inlet Pressure Transducer Alarm Delay" %
%   N7:77  OPEN_PX1_WRN_DLY  "CONFIG Gas Inlet Pressure Transducer Warning Delay" %
%   B26:2/0  OPEN_PX1_ALM_EN  "CONFIG Gas Inlet Pressure Transmitter Alarm Enable" %
%   B26:7/0  OPEN_PX1_WRN_EN  "CONFIG Gas Inlet Pressure Transmitter Warning Enable" %

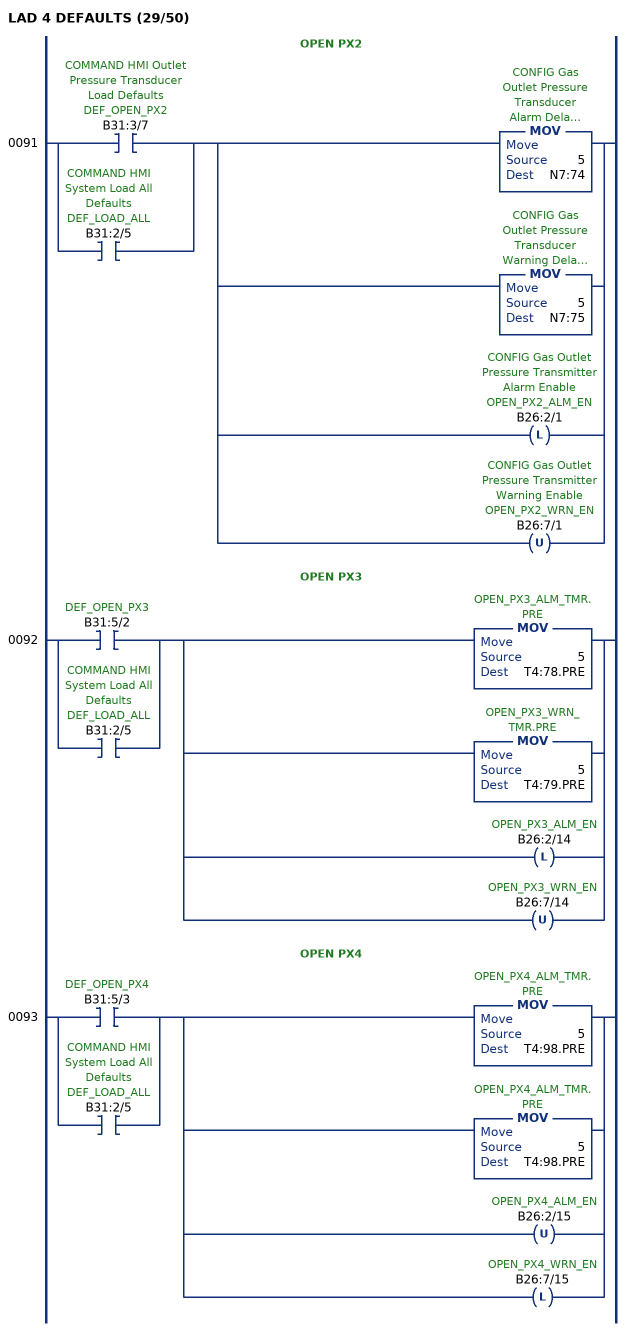
% Rung: 91 %
% TITLE: OPEN PX2 %
SOR BST XIC B31:3/7 NXB XIC B31:2/5 BND BST MOV 5 N7:74 NXB MOV 5 N7:75 NXB OTL B26:2/1 NXB OTU B26:7/1 BND EOR
%   B31:3/7  DEF_OPEN_PX2  "COMMAND HMI Outlet Pressure Transducer Load Defaults" %
%   B31:2/5  DEF_LOAD_ALL  "COMMAND HMI System Load All Defaults" %
%   N7:74  OPEN_PX2_ALM_DLY  "CONFIG Gas Outlet Pressure Transducer Alarm Delay" %
%   N7:75  OPEN_PX2_WRN_DLY  "CONFIG Gas Outlet Pressure Transducer Warning Delay" %
%   B26:2/1  OPEN_PX2_ALM_EN  "CONFIG Gas Outlet Pressure Transmitter Alarm Enable" %
%   B26:7/1  OPEN_PX2_WRN_EN  "CONFIG Gas Outlet Pressure Transmitter Warning Enable" %
% Rung: 92 %
% TITLE: OPEN PX3 %
SOR BST XIC B31:5/2 NXB XIC B31:2/5 BND BST MOV 5 T4:78.PRE NXB MOV 5 T4:79.PRE NXB OTL B26:2/14 NXB OTU B26:7/14 BND EOR
%   B31:5/2  DEF_OPEN_PX3 %
%   B31:2/5  DEF_LOAD_ALL  "COMMAND HMI System Load All Defaults" %
%   T4:78  OPEN_PX3_ALM_TMR %
%   T4:79  OPEN_PX3_WRN_TMR %
%   B26:2/14  OPEN_PX3_ALM_EN %
%   B26:7/14  OPEN_PX3_WRN_EN %
% Rung: 93 %
% TITLE: OPEN PX4 %
SOR BST XIC B31:5/3 NXB XIC B31:2/5 BND BST MOV 5 T4:98.PRE NXB MOV 5 T4:98.PRE NXB OTU B26:2/15 NXB OTL B26:7/15 BND EOR
%   B31:5/3  DEF_OPEN_PX4 %
%   B31:2/5  DEF_LOAD_ALL  "COMMAND HMI System Load All Defaults" %
%   T4:98  OPEN_PX4_ALM_TMR %
%   B26:2/15  OPEN_PX4_ALM_EN %
%   B26:7/15  OPEN_PX4_WRN_EN %

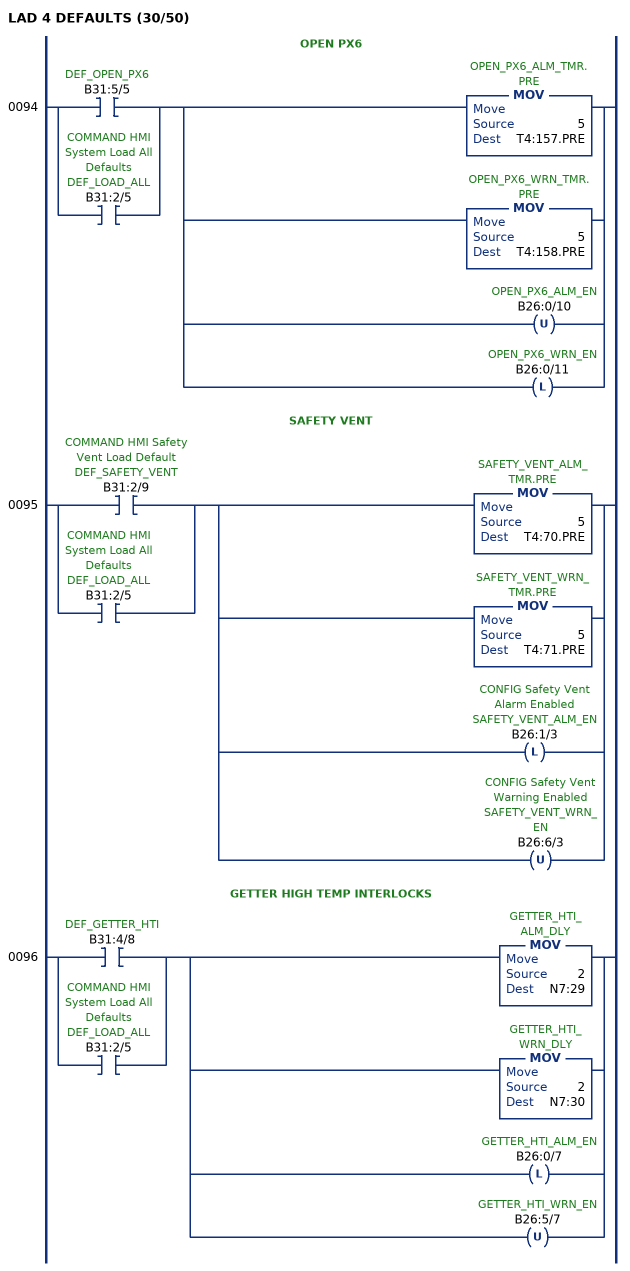
% Rung: 94 %
% TITLE: OPEN PX6 %
SOR BST XIC B31:5/5 NXB XIC B31:2/5 BND BST MOV 5 T4:157.PRE NXB MOV 5 T4:158.PRE NXB OTU B26:0/10 NXB OTL B26:0/11 BND EOR
%   B31:5/5  DEF_OPEN_PX6 %
%   B31:2/5  DEF_LOAD_ALL  "COMMAND HMI System Load All Defaults" %
%   T4:157  OPEN_PX6_ALM_TMR %
%   T4:158  OPEN_PX6_WRN_TMR %
%   B26:0/10  OPEN_PX6_ALM_EN %
%   B26:0/11  OPEN_PX6_WRN_EN %
% Rung: 95 %
% TITLE: SAFETY VENT %
SOR BST XIC B31:2/9 NXB XIC B31:2/5 BND BST MOV 5 T4:70.PRE NXB MOV 5 T4:71.PRE NXB OTL B26:1/3 NXB OTU B26:6/3 BND EOR
%   B31:2/9  DEF_SAFETY_VENT  "COMMAND HMI Safety Vent Load Default" %
%   B31:2/5  DEF_LOAD_ALL  "COMMAND HMI System Load All Defaults" %
%   T4:70  SAFETY_VENT_ALM_TMR %
%   T4:71  SAFETY_VENT_WRN_TMR %
%   B26:1/3  SAFETY_VENT_ALM_EN  "CONFIG Safety Vent Alarm Enabled" %
%   B26:6/3  SAFETY_VENT_WRN_EN  "CONFIG Safety Vent Warning Enabled" %
% Rung: 96 %
% TITLE: GETTER HIGH TEMP INTERLOCKS %
SOR BST XIC B31:4/8 NXB XIC B31:2/5 BND BST MOV 2 N7:29 NXB MOV 2 N7:30 NXB OTL B26:0/7 NXB OTU B26:5/7 BND EOR
%   B31:4/8  DEF_GETTER_HTI %
%   B31:2/5  DEF_LOAD_ALL  "COMMAND HMI System Load All Defaults" %
%   N7:29  GETTER_HTI_ALM_DLY %
%   N7:30  GETTER_HTI_WRN_DLY %
%   B26:0/7  GETTER_HTI_ALM_EN %
%   B26:5/7  GETTER_HTI_WRN_EN %

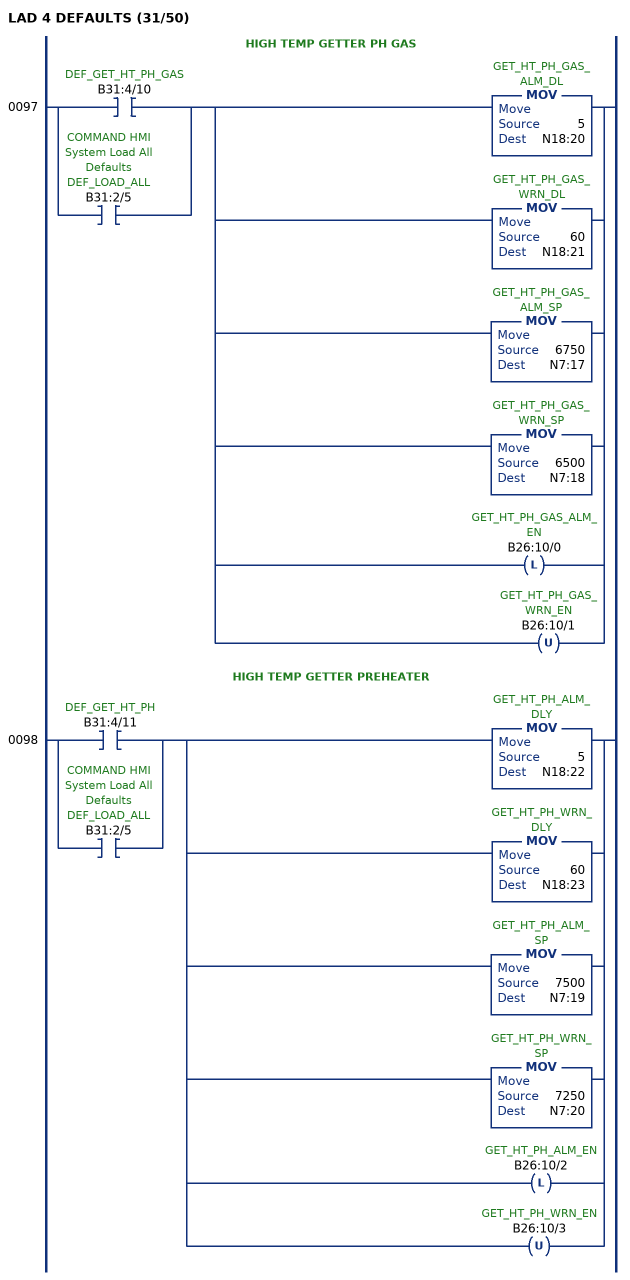
% Rung: 97 %
% TITLE: HIGH TEMP GETTER PH GAS %
SOR BST XIC B31:4/10 NXB XIC B31:2/5 BND BST MOV 5 N18:20 NXB MOV 60 N18:21 NXB MOV 6750 N7:17 NXB MOV 6500 N7:18 NXB OTL B26:10/0 NXB OTU B26:10/1 BND EOR
%   B31:4/10  DEF_GET_HT_PH_GAS %
%   B31:2/5  DEF_LOAD_ALL  "COMMAND HMI System Load All Defaults" %
%   N18:20  GET_HT_PH_GAS_ALM_DL %
%   N18:21  GET_HT_PH_GAS_WRN_DL %
%   N7:17  GET_HT_PH_GAS_ALM_SP %
%   N7:18  GET_HT_PH_GAS_WRN_SP %
%   B26:10/0  GET_HT_PH_GAS_ALM_EN %
%   B26:10/1  GET_HT_PH_GAS_WRN_EN %
% Rung: 98 %
% TITLE: HIGH TEMP GETTER PREHEATER %
SOR BST XIC B31:4/11 NXB XIC B31:2/5 BND BST MOV 5 N18:22 NXB MOV 60 N18:23 NXB MOV 7500 N7:19 NXB MOV 7250 N7:20 NXB OTL B26:10/2 NXB OTU B26:10/3 BND EOR
%   B31:4/11  DEF_GET_HT_PH %
%   B31:2/5  DEF_LOAD_ALL  "COMMAND HMI System Load All Defaults" %
%   N18:22  GET_HT_PH_ALM_DLY %
%   N18:23  GET_HT_PH_WRN_DLY %
%   N7:19  GET_HT_PH_ALM_SP %
%   N7:20  GET_HT_PH_WRN_SP %
%   B26:10/2  GET_HT_PH_ALM_EN %
%   B26:10/3  GET_HT_PH_WRN_EN %

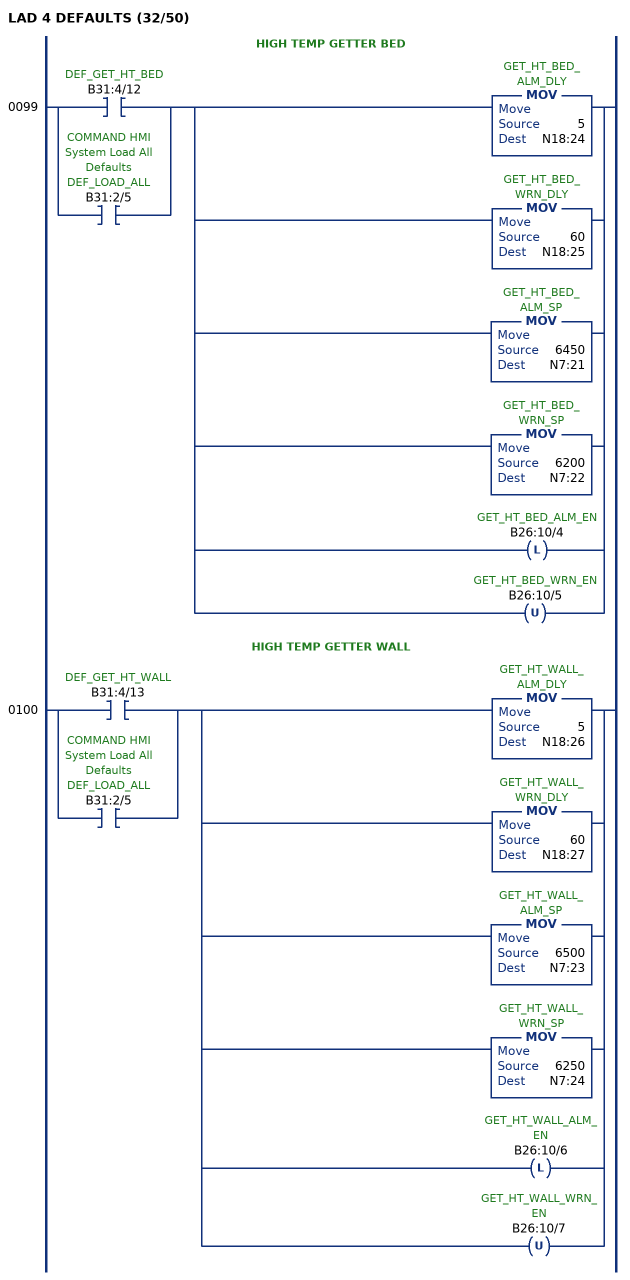
% Rung: 99 %
% TITLE: HIGH TEMP GETTER BED %
SOR BST XIC B31:4/12 NXB XIC B31:2/5 BND BST MOV 5 N18:24 NXB MOV 60 N18:25 NXB MOV 6450 N7:21 NXB MOV 6200 N7:22 NXB OTL B26:10/4 NXB OTU B26:10/5 BND EOR
%   B31:4/12  DEF_GET_HT_BED %
%   B31:2/5  DEF_LOAD_ALL  "COMMAND HMI System Load All Defaults" %
%   N18:24  GET_HT_BED_ALM_DLY %
%   N18:25  GET_HT_BED_WRN_DLY %
%   N7:21  GET_HT_BED_ALM_SP %
%   N7:22  GET_HT_BED_WRN_SP %
%   B26:10/4  GET_HT_BED_ALM_EN %
%   B26:10/5  GET_HT_BED_WRN_EN %
% Rung: 100 %
% TITLE: HIGH TEMP GETTER WALL %
SOR BST XIC B31:4/13 NXB XIC B31:2/5 BND BST MOV 5 N18:26 NXB MOV 60 N18:27 NXB MOV 6500 N7:23 NXB MOV 6250 N7:24 NXB OTL B26:10/6 NXB OTU B26:10/7 BND EOR
%   B31:4/13  DEF_GET_HT_WALL %
%   B31:2/5  DEF_LOAD_ALL  "COMMAND HMI System Load All Defaults" %
%   N18:26  GET_HT_WALL_ALM_DLY %
%   N18:27  GET_HT_WALL_WRN_DLY %
%   N7:23  GET_HT_WALL_ALM_SP %
%   N7:24  GET_HT_WALL_WRN_SP %
%   B26:10/6  GET_HT_WALL_ALM_EN %
%   B26:10/7  GET_HT_WALL_WRN_EN %

